{attribute addProperty BoxType "IODEVICETYPE_ETHERCATPROT"}
{attribute addProperty Id "Beckhoff_ELM3xxxBeckhoff_ELM3xxx_445FD47E2992374Beckhoff_ELM31xxBeckhoff_ELM31xx_D2520EAD82081026Beckhoff_ELM35xxBeckhoff_ELM35xx_750E8EE93344418Beckhoff_ELM36xxBeckhoff_ELM36xx_314CE8BD4176522Beckhoff_ELM37xxBeckhoff_ELM37xx_58D302163952494Beckhoff_ELM3xxx_0030Beckhoff_ELM3xxx_0030_079858E12512314Beckhoff_ELM9xxxBeckhoff_ELM9xxx_07C3C7BE2826353.25SyncUnitsSyncUnits_3FA29F3C21627InputsInputs_C75D3FEC1280160OutputsOutputs_47D1E803848106InfoDataInfoData_45F98C5022428"}
{attribute addProperty CRC "548046093"}
{attribute addProperty SizeInBites "30578"}
{attribute addProperty SizeInBytes "3822.25"}
TYPE EtherCAT_Master_ELMxxxx_20AA850D :
STRUCT
	{attribute addProperty Name "Beckhoff_ELM3xxx"}
	Beckhoff_ELM3xxx : Beckhoff_ELM3xxx_445FD47E;
	{attribute addProperty Name "Beckhoff_ELM31xx"}
	Beckhoff_ELM31xx : Beckhoff_ELM31xx_D2520EAD;
	{attribute addProperty Name "Beckhoff_ELM35xx"}
	Beckhoff_ELM35xx : Beckhoff_ELM35xx_750E8EE9;
	{attribute addProperty Name "Beckhoff_ELM36xx"}
	Beckhoff_ELM36xx : Beckhoff_ELM36xx_314CE8BD;
	{attribute addProperty Name "Beckhoff_ELM37xx"}
	Beckhoff_ELM37xx : Beckhoff_ELM37xx_58D30216;
	{attribute addProperty Name "Beckhoff_ELM3xxx_0030"}
	Beckhoff_ELM3xxx_0030 : Beckhoff_ELM3xxx_0030_079858E1;
	{attribute addProperty Name "Beckhoff_ELM9xxx"}
	Beckhoff_ELM9xxx : Beckhoff_ELM9xxx_07C3C7BE;
	{attribute addProperty Name "SyncUnits"}
	SyncUnits : SyncUnits_3FA29F3C;
	{attribute addProperty Name "Inputs"}
	Inputs : Inputs_C75D3FEC;
	{attribute addProperty Name "Outputs"}
	Outputs : Outputs_47D1E803;
	{attribute addProperty Name "InfoData"}
	InfoData : InfoData_45F98C50;
END_STRUCT
END_TYPE

(* stored: Version 1.2.0.0, ProductVersion 3.1.4024.9
   DUT EtherCAT_Master_ELMxxxx_20AA850D: Id {7a411733-5ede-4ec5-9e2b-1fc8af9d8f91} *)
